FUNCTION_BLOCK FB_GatewaySmokeTests EXTENDS TcUnit.FB_TestSuite

GatewayCanExecuteTcUnit();

GatewayReportsFailedTcUnit();

METHOD PRIVATE GatewayCanExecuteTcUnit
TEST('GatewayCanExecuteTcUnit');
AssertTrue(
    Condition := TRUE,
    Message := 'Gateway TcUnit smoke test should pass');
TEST_FINISHED();
END_METHOD

METHOD PRIVATE GatewayReportsFailedTcUnit
TEST('GatewayReportsFailedTcUnit');
AssertTrue(
    Condition := FALSE,
    Message := 'Intentional gateway TcUnit failure scenario');
TEST_FINISHED();
END_METHOD

END_FUNCTION_BLOCK

(* stored: Version 1.1.0.1, ProductVersion 3.1.4024.9
   POU FB_GatewaySmokeTests: Id {7794579c-f33b-4b1c-9bd6-31230f87ed8f}, SpecialFunc None
   Method GatewayCanExecuteTcUnit: Id {fededc5f-649e-4cf5-a82c-0bb8d8ea29f8}
   Method GatewayReportsFailedTcUnit: Id {fb286950-5673-4e6e-b82d-69d6d8a1ae51} *)
